FUNCTION_BLOCK Logger
VAR_INPUT
	bExecute : BOOL;
	sPathName : STRING;
END_VAR
VAR_OUTPUT
END_VAR
VAR
	aBuffer : ARRAY[1..cMaxBufferRange] OF T_MaxString;
	aWorkBuffer : ARRAY[1..cMaxBufferRange] OF T_MaxString;
	aEmptyBuffer : ARRAY[1..cMaxBufferRange] OF T_MaxString; 
	
	fbFileWrite : FB_FileWrite;
	udiBufferCounter : UDINT;
	udiWorkCounter : UDINT;
	hFile : UINT;	
	
	fbFileOpen : FB_FileOpen;
	fbFilePuts : FB_FilePuts;
	fbFileClose : FB_FileClose;
	
	fbGetSystemTime : GETSYSTEMTIME;
	fbRepeatTimer : TON;
	diStep  : DINT;
	i : UDINT;
	bFilePutsIdle : BOOL;
	bExecuteFilePuts : BOOL;
	bInit : BOOL;
END_VAR
VAR CONSTANT
	cMaxBufferRange : UDINT := 1000;
END_VAR

fbFileOpen(
	sNetId:= , 
	sPathName:= sPathName,
	nMode:= FOPEN_MODEAPPEND OR FOPEN_MODETEXT, 
	ePath:= , 
	bExecute:=, 
	tTimeout:= , 
	bBusy=> , 
	bError=> , 
	nErrId=> , 
	hFile=> hFile);

fbFileWrite(
	sNetId:= , 
	hFile:= hFile, 
	pWriteBuff:= ADR(aWorkBuffer) , 
	cbWriteLen:= , 
	bExecute:= , 
	tTimeout:= , 
	bBusy=> , 
	bError=> , 
	nErrId=> , 
	cbWrite=> );

fbFileClose(
	sNetId:= , 
	hFile:= hFile, 
	bExecute:= , 
	tTimeout:= , 
	bBusy=> , 
	bError=> , 
	nErrId=> );
	
fbRepeatTimer(IN:= , PT:= T#2S, Q=> , ET=> );
//fbTime();

IF NOT bInit
THEN
	bInit := TRUE;
	FOR i := 1 TO cMaxBufferRange DO
		aEmptyBuffer[i] := '';
		aBuffer[i] := '';
		aWorkBuffer[i] := '';
	END_FOR
END_IF

IF 			bExecute
	AND  	diStep = 0
THEN
	diStep := 10;
END_IF	

CASE diStep OF
	
	10:
	
		fbFileOpen.bExecute := TRUE;
		fbRepeatTimer.IN := TRUE;
		diStep := 20;
		
	20:
	
		IF 		NOT fbFileOpen.bBusy
			AND NOT fbFIleOpen.bError
		THEN
			fbFileOpen.bExecute := FALSE;
			diStep := 30;
		END_IF
		
	30:
		
		IF udiBufferCounter > 0
		THEN
			udiWorkCounter := udiBufferCounter;
			udiBufferCounter := 0;
			
			aWorkBuffer := aBuffer;
			aBuffer := aEmptyBuffer;
			
			fbFileWrite.cbWriteLen := udiWorkCounter * (SIZEOF(T_MaxString));
			fbFileWrite.bExecute := TRUE;
			
			diStep := 40;
		ELSIF NOT bExecute
		THEN
			diStep := 50;
		END_IF
		
		
	40:
		
		IF NOT fbFileWrite.bBusy
		THEN
			
			fbFileWrite.bExecute := FALSE;
			IF fbRepeatTimer.Q
			THEN
				fbRepeatTImer.IN := FALSE;
				diStep := 50;
			ELSE
				diStep := 30;
			END_IF
			
		END_IF
		
	50:
	
		fbFileClose.bExecute := TRUE;
		diStep := 60;
		
	60: 
	
		IF 		NOT fbFileClose.bBusy
			AND NOT fbFileClose.bError
		THEN
			fbFileClose.bExecute := FALSE;
			IF bExecute 
			THEN
				
				diStep := 10;
			ELSE
				diStep := 0;
			END_IF
			
		END_IF
	
END_CASE

METHOD Write 
VAR_INPUT
	sMessage : T_MaxString;
END_VAR
VAR
	iLen : INT;
	iFillNumber : INT;
	i : INT;
	sTime : STRING;
	fileTime        : T_FILETIME;
END_VAR
IF udiBufferCounter < cMaxBufferRange
THEN

	udiBufferCounter := udiBufferCounter + 1;
	
	fbGetSystemTime(timeLoDW=>fileTime.dwLowDateTime, timeHiDW=>fileTime.dwHighDateTime );
	sTime :=SYSTEMTIME_TO_STRING( FILETIME_TO_SYSTEMTIME( fileTime ) );
	
	aBuffer[udiBufferCounter] := sTime;
	aBuffer[udiBufferCounter] := CONCAT(aBuffer[udiBufferCounter],': ');
	aBuffer[udiBufferCounter] := CONCAT(aBuffer[udiBufferCounter],sMessage);
	
	iLen := LEN(aBuffer[udiBufferCounter]);
	iFillNumber := 254-iLen;
	
	FOR i := 1 TO iFillNumber DO
		aBuffer[udiBufferCounter] := CONCAT(aBuffer[udiBufferCounter],' ');
	END_FOR
	
	aBuffer[udiBufferCounter][255] := F_ToAsc('$N');
	
END_IF
END_METHOD

END_FUNCTION_BLOCK

(* stored: Version 1.1.0.1, ProductVersion 3.1.4024.2
   POU Logger: Id {2299ad2c-33aa-48d7-80de-77920f3a5952}, SpecialFunc None
   Method Write: Id {39218833-d461-4ffc-9b85-e53207615746} *)
